FUNCTION_BLOCK LinksRechts_AX (* Basic FB with Links-Rechts, with AX Adapter *)
  (* Standard: 61499-2; Description: Copyright (c) 2025 HR Agrartechnik GmbH This program and the accompanying materials are made available under the terms of the Eclipse Public License 2.0 which is available at https://www.eclipse.org/legal/epl-2.0/ SPDX-License-Identifier: EPL-2.0 Nur Rechtslauf ist vorrangig vor Nur Linkslauf. *)
  (* Version 1.1, 2026-01-16, Gemini, HR Agrartechnik GmbH *)
  PACKAGE logiBUS::utils::sequence::verteiler;
  IMPORT eclipse4diac::core::TypeHash;
  IMPORT logiBUS::utils::sequence::verteiler::LinksRechts::STATES;
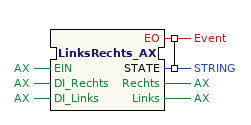
  EVENT_OUTPUT
    EO WITH STATE;
  END_EVENT
  VAR_OUTPUT
    STATE : STRING;
  END_VAR
  SOCKETS
    EIN : adapter::types::unidirectional::AX; (* Einschalten *)
    DI_Rechts : adapter::types::unidirectional::AX; (* Nur Rechtslauf *)
    DI_Links : adapter::types::unidirectional::AX; (* Nur Linkslauf *)
  END_SOCKETS
  PLUGS
    Rechts : adapter::types::unidirectional::AX; (* Rechtslauf *)
    Links : adapter::types::unidirectional::AX; (* Linkslauf *)
  END_PLUGS
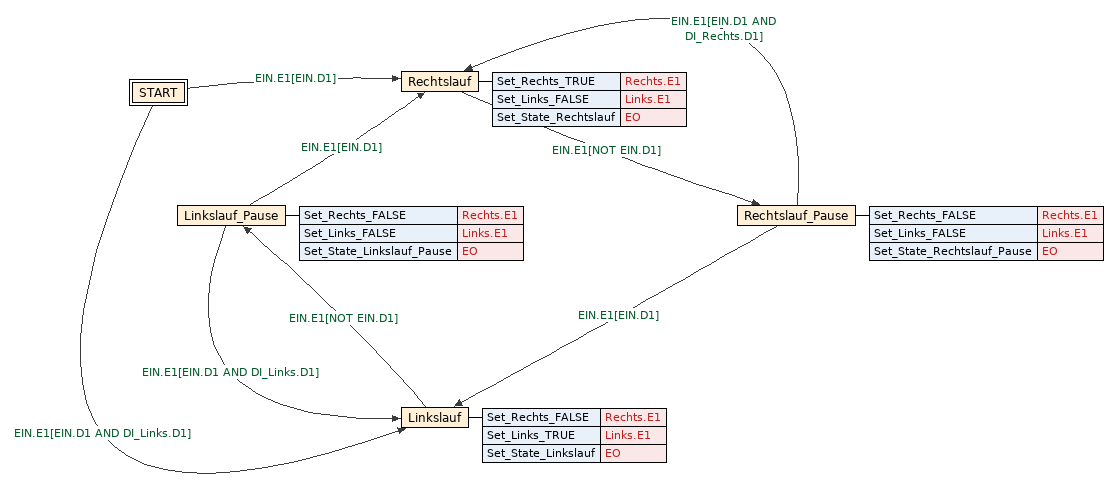
  EC_STATES
    START; (* Initial State *)
    Rechtslauf : Set_Rechts_TRUE -> Rechts.E1, Set_Links_FALSE -> Links.E1, Set_State_Rechtslauf -> EO;
    Rechtslauf_Pause : Set_Rechts_FALSE -> Rechts.E1, Set_Links_FALSE -> Links.E1, Set_State_Rechtslauf_Pause -> EO;
    Linkslauf : Set_Rechts_FALSE -> Rechts.E1, Set_Links_TRUE -> Links.E1, Set_State_Linkslauf -> EO;
    Linkslauf_Pause : Set_Rechts_FALSE -> Rechts.E1, Set_Links_FALSE -> Links.E1, Set_State_Linkslauf_Pause -> EO;
  END_STATES
  EC_TRANSITIONS
    START TO Linkslauf := EIN.E1[EIN.D1 AND DI_Links.D1];
    START TO Rechtslauf := EIN.E1[EIN.D1];
    Rechtslauf TO Rechtslauf_Pause := EIN.E1[NOT EIN.D1];
    Rechtslauf_Pause TO Rechtslauf := EIN.E1[EIN.D1 AND DI_Rechts.D1];
    Rechtslauf_Pause TO Linkslauf := EIN.E1[EIN.D1];
    Linkslauf TO Linkslauf_Pause := EIN.E1[NOT EIN.D1];
    Linkslauf_Pause TO Linkslauf := EIN.E1[EIN.D1 AND DI_Links.D1];
    Linkslauf_Pause TO Rechtslauf := EIN.E1[EIN.D1];
  END_TRANSITIONS
  ALGORITHM Set_Rechts_TRUE IN ST:
Rechts.D1 := BOOL#TRUE;
  END_ALGORITHM
  ALGORITHM Set_Rechts_FALSE IN ST:
Rechts.D1 := BOOL#FALSE;
  END_ALGORITHM
  ALGORITHM Set_Links_TRUE IN ST:
Links.D1 := BOOL#TRUE;
  END_ALGORITHM
  ALGORITHM Set_Links_FALSE IN ST:
Links.D1 := BOOL#FALSE;
  END_ALGORITHM
  ALGORITHM Set_State_Rechtslauf IN ST:
STATE := STATES::Rechtslauf;
  END_ALGORITHM
  ALGORITHM Set_State_Linkslauf IN ST:
STATE := STATES::Linkslauf;
  END_ALGORITHM
  ALGORITHM Set_State_Rechtslauf_Pause IN ST:
STATE := STATES::Rechtslauf_Pause;
  END_ALGORITHM
  ALGORITHM Set_State_Linkslauf_Pause IN ST:
STATE := STATES::Linkslauf_Pause;
  END_ALGORITHM
END_FUNCTION_BLOCK
